// Mitsubishi GX Works2 project: q04   PLC: Q02/Q02H

PROGRAM MAIN
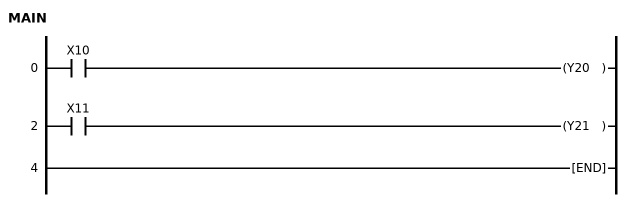
0     LD      X10
      OUT     Y20
2     LD      X11
      OUT     Y21
4     END
END_PROGRAM

PROGRAM touth
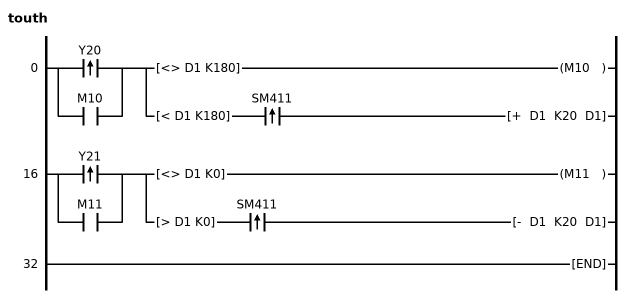
0     LDP     Y20
      OR      M10
      MPS
      AND<>   D1 K180
      OUT     M10
      MPP
      AND<    D1 K180
      ANDP    SM411
      +       D1 K20 D1
16    LDP     Y21
      OR      M11
      MPS
      AND<>   D1 K0
      OUT     M11
      MPP
      AND>    D1 K0
      ANDP    SM411
      -       D1 K20 D1
32    END
END_PROGRAM
